(* Logix 5000 project; controller IronPelletsFactory Emulate 5570 rev 30.12; software revision 30.02 *)
// A program for the materials delivery equipment of the iron process.

TASK MainTask (continuous, watchdog 500 ms) : MainProgram

MODULES
   Local : Emulate 5570 (ICP 2, rev 30.12)
      Simulate_IO3 : vendor 1 type 0 code 15 (ICP 3, rev 1.1, Output RPI 50 ms)
      Simulate_IO4 : vendor 1 type 0 code 15 (ICP 4, rev 1.1, Output RPI 50 ms)
END_MODULES

VAR_GLOBAL   (* controller tags *)
   CarPositionONS : BOOL;
   CokeGateFault : BOOL;
   CokeGateFaultBit0 : BOOL := 1;
   CokeGateFaultBit1 : BOOL;
   CokeGateFaultTimer : TIMER := (PRE := 10000);   // Times how long the coke gate has been open or closed.
   Furnace : DINT;
   MaterialsPresent : BOOL := 1;
   NumberOfLoads : DINT := 20;   // This is how many times you have to load the scale car to fill the furnace to its target weight.
   PelletGateFault : BOOL;
   PelletGateFaultBit0 : BOOL := 1;
   PelletGateFaultBit1 : BOOL;
   PelletGateFaultTimer : TIMER := (PRE := 10000);   // Times how long the pellet gate has been open or closed.
   ScaleInRange : BOOL;
   SimFillTime : TIMER := (PRE := 1000);   // Times how long it takes to fill the car.
   SystemCommandONS : BOOL := 1;
   WeightLoad : DINT := 4000;
   WeightTotal : DINT := 80000;
END_VAR

PROGRAM MainProgram   (* main routine MainRoutine *)
VAR
   CarPosition : ALIAS FOR Local:3:I.Data[0].12;
   CokeConveyorOut : ALIAS FOR Local:4:O.Data[0].3;
   CokeGateOut : ALIAS FOR Local:4:O.Data[0].1;
   CokeHigh : ALIAS FOR Local:3:I.Data[0].1;
   CokeLow : ALIAS FOR Local:3:I.Data[0].9;
   PelletGateOut : ALIAS FOR Local:4:O.Data[0].4;
   Start : ALIAS FOR Local:3:I.Data[0].0;
   Stop : ALIAS FOR Local:3:I.Data[0].8;
   SystemCommand : ALIAS FOR Local:4:O.Data[0].0;
   Weight : DINT := 9;   // The weight of the weigh scale.
   WeightTarget : ALIAS FOR Local:3:I.Data[0].13;
END_VAR
VAR_INPUT
   SimWeight : DINT;
END_VAR

ROUTINE Coke_Conveyor   (* ladder *)
// Refills the stockhouse with coke whenever it gets low.
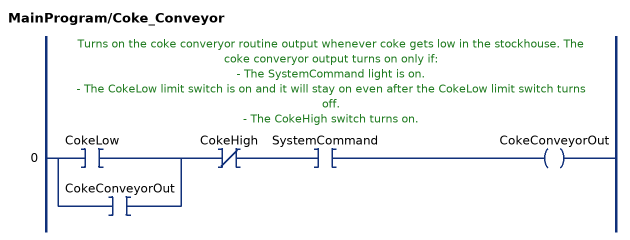
   // Turns on the coke converyor routine output whenever coke gets low in the stockhouse. The coke converyor output turns on only if:
   // - The SystemCommand light is on.
   // - The CokeLow limit switch is on and it will stay on even after the CokeLow limit switch turns off.
   // - The CokeHigh switch turns on.
   0: [XIC(CokeLow) ,XIC(CokeConveyorOut) ]XIO(CokeHigh)XIC(SystemCommand)OTE(CokeConveyorOut);
END_ROUTINE

ROUTINE MainRoutine   (* ladder *)
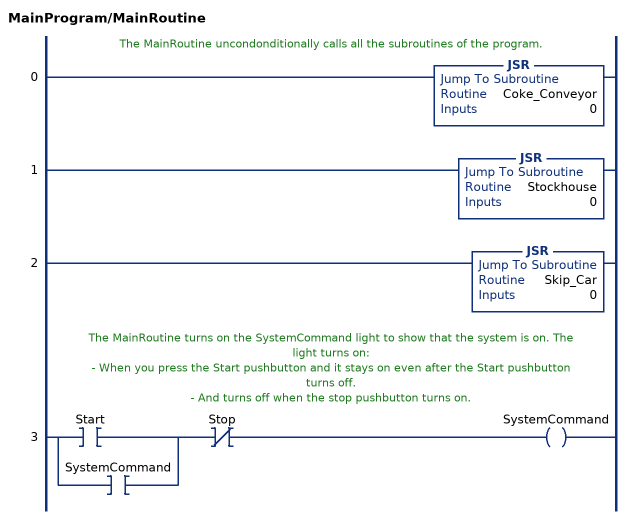
   // The MainRoutine uncondonditionally calls all the subroutines of the program.
   0: JSR(Coke_Conveyor,0);
   1: JSR(Stockhouse,0);
   2: JSR(Skip_Car,0);
   // The MainRoutine turns on the SystemCommand light to show that the system is on. The light turns on:
   // - When you press the Start pushbutton and it stays on even after the Start pushbutton turns off.
   // - And turns off when the stop pushbutton turns on.
   3: [XIC(Start) ,XIC(SystemCommand) ]XIO(Stop)OTE(SystemCommand);
END_ROUTINE

ROUTINE Skip_Car   (* ladder *)
// Delivers coke and iron pellets to top of the furnace.
END_ROUTINE

ROUTINE Stockhouse   (* ladder *)
// Measures set weights of coke and iron pellets and delivers them to the skip car.
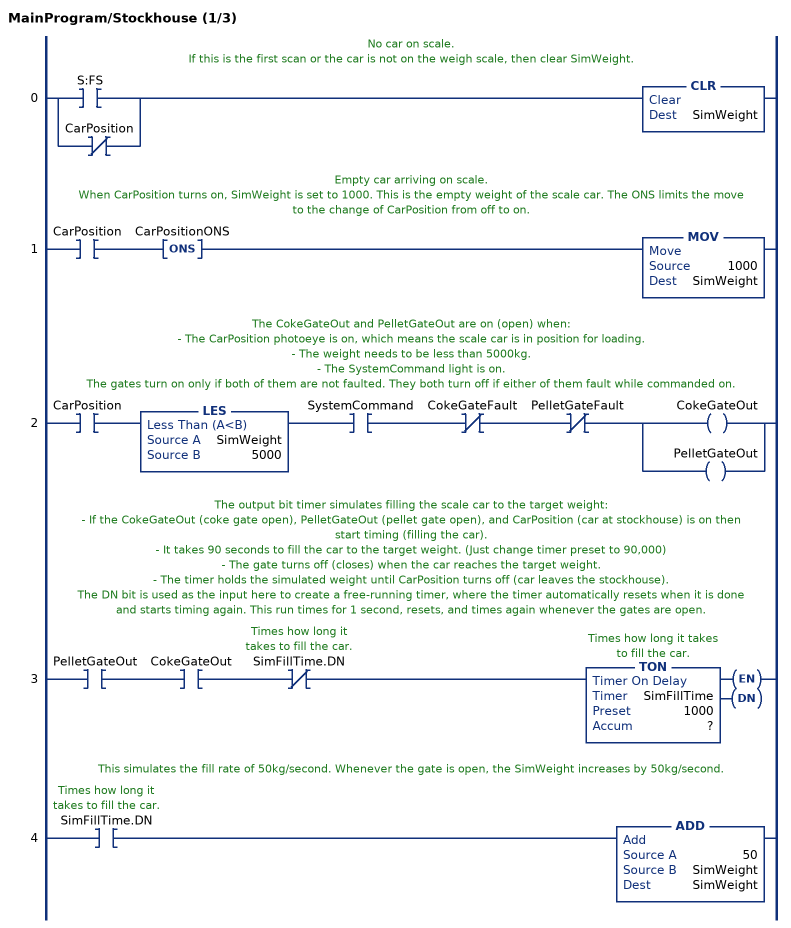
   // No car on scale.
   // If this is the first scan or the car is not on the weigh scale, then clear SimWeight.
   0: [XIC(S:FS) ,XIO(CarPosition) ]CLR(SimWeight);
   // Empty car arriving on scale.
   // When CarPosition turns on, SimWeight is set to 1000. This is the empty weight of the scale car. The ONS limits the move to the change of CarPosition from off to on.
   1: XIC(CarPosition)ONS(CarPositionONS)MOV(1000,SimWeight);
   // The CokeGateOut and PelletGateOut are on (open) when:
   // - The CarPosition photoeye is on, which means the scale car is in position for loading.
   // - The weight needs to be less than 5000kg.
   // - The SystemCommand light is on.
   // The gates turn on only if both of them are not faulted. They both turn off if either of them fault while commanded on.
   2: XIC(CarPosition)LES(SimWeight,5000)XIC(SystemCommand)XIO(CokeGateFault)XIO(PelletGateFault)[OTE(CokeGateOut) ,OTE(PelletGateOut) ];
   // The output bit timer simulates filling the scale car to the target weight:
   // - If the CokeGateOut (coke gate open), PelletGateOut (pellet gate open), and CarPosition (car at stockhouse) is on then start timing (filling the car).
   // - It takes 90 seconds to fill the car to the target weight. (Just change timer preset to 90,000)
   // - The gate turns off (closes) when the car reaches the target weight.
   // - The timer holds the simulated weight until CarPosition turns off (car leaves the stockhouse).
   // The DN bit is used as the input here to create a free-running timer, where the timer automatically resets when it is done and starts timing again. This run times for 1 second, resets, and times again whenever the gates are open.
   3: XIC(PelletGateOut)XIC(CokeGateOut)XIO(SimFillTime.DN)TON(SimFillTime,?,?);
   // This simulates the fill rate of 50kg/second. Whenever the gate is open, the SimWeight increases by 50kg/second.
   4: XIC(SimFillTime.DN)ADD(50,SimWeight,SimWeight);
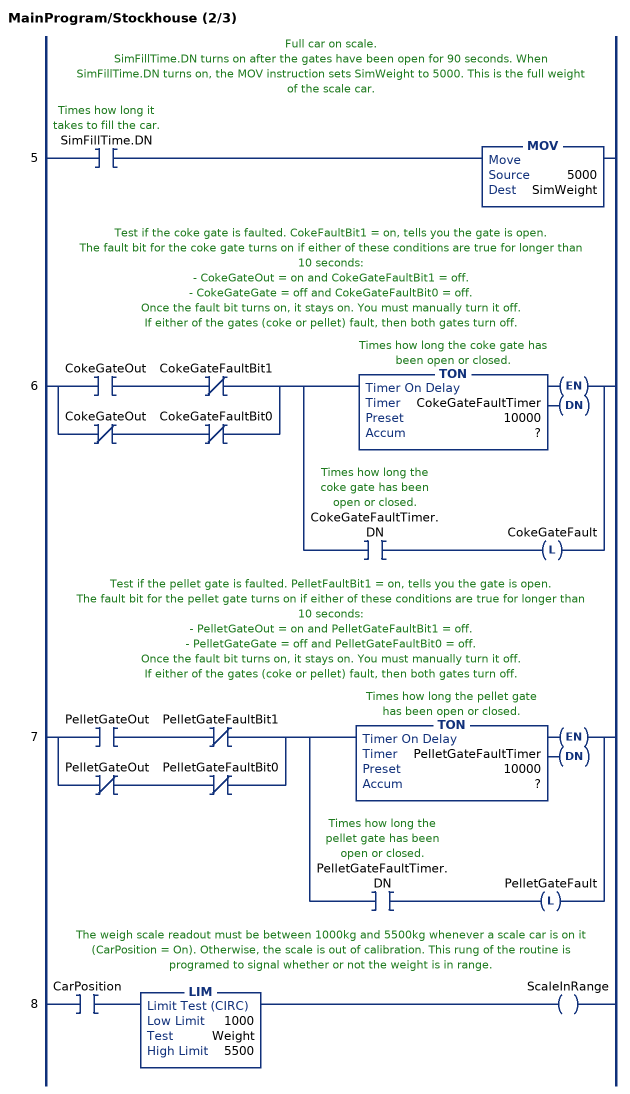
   // Full car on scale.
   // SimFillTime.DN turns on after the gates have been open for 90 seconds. When SimFillTime.DN turns on, the MOV instruction sets SimWeight to 5000. This is the full weight of the scale car.
   5: XIC(SimFillTime.DN)MOV(5000,SimWeight);
   // Test if the coke gate is faulted. CokeFaultBit1 = on, tells you the gate is open.
   // The fault bit for the coke gate turns on if either of these conditions are true for longer than 10 seconds:
   // - CokeGateOut = on and CokeGateFaultBit1 = off.
   // - CokeGateGate = off and CokeGateFaultBit0 = off.
   // Once the fault bit turns on, it stays on. You must manually turn it off.
   // If either of the gates (coke or pellet) fault, then both gates turn off.
   6: [XIC(CokeGateOut) XIO(CokeGateFaultBit1) ,XIO(CokeGateOut) XIO(CokeGateFaultBit0) ][TON(CokeGateFaultTimer,?,?) ,XIC(CokeGateFaultTimer.DN) OTL(CokeGateFault) ];
   // Test if the pellet gate is faulted. PelletFaultBit1 = on, tells you the gate is open.
   // The fault bit for the pellet gate turns on if either of these conditions are true for longer than 10 seconds:
   // - PelletGateOut = on and PelletGateFaultBit1 = off.
   // - PelletGateGate = off and PelletGateFaultBit0 = off.
   // Once the fault bit turns on, it stays on. You must manually turn it off.
   // If either of the gates (coke or pellet) fault, then both gates turn off.
   7: [XIC(PelletGateOut) XIO(PelletGateFaultBit1) ,XIO(PelletGateOut) XIO(PelletGateFaultBit0) ][TON(PelletGateFaultTimer,?,?) ,XIC(PelletGateFaultTimer.DN) OTL(PelletGateFault) ];
   // The weigh scale readout must be between 1000kg and 5500kg whenever a scale car is on it (CarPosition = On). Otherwise, the scale is out of calibration. This rung of the routine is programed to signal whether or not the weight is in range.
   8: XIC(CarPosition)LIM(1000,Weight,5500)OTE(ScaleInRange);
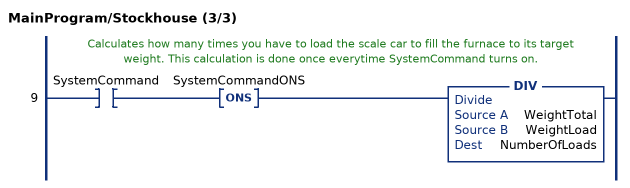
   // Calculates how many times you have to load the scale car to fill the furnace to its target weight. This calculation is done once everytime SystemCommand turns on.
   9: XIC(SystemCommand)ONS(SystemCommandONS)DIV(WeightTotal,WeightLoad,NumberOfLoads);
END_ROUTINE
END_PROGRAM
